PROGRAM MAIN
VAR
END_VAR

END_PROGRAM

(* stored: Version 1.1.0.1
   POU MAIN: Id {d7bd07a9-632a-4512-a44e-2ca193c0ff70} *)
